// TIA Portal V20 export
VAR_GLOBAL   // PLC tag table "Unit1Em12"
   "BA060ZSIBK18.00" AT %I1068.0 : Bool;   // (HOME) WEIGHT NG CLAMP MOVER OPEN
   "BA060ZSIBK18.01" AT %I1068.1 : Bool;   // (HOME) WEIGHT NG CLAMP LEFT OPEN
   "BA060ZSIBK18.02" AT %I1068.2 : Bool;   // (HOME) WEIGHT NG CLAMP RIGHT OPEN
   "BA060ZSIBK18.03" AT %I1068.3 : Bool;   // (HOME) WEIGHT NG CLAMP Z-AXIS UP
   "BA060ZSIBK18.04" AT %I1068.4 : Bool;   // (HOME) WEIGHT NG CLAMP MOVER BACKWARD
   "BA060ZSIBK18.05" AT %I1068.5 : Bool;   // (HOME) WEIGHT NG BOX LIFT DOWN
   "BA060ZSIBK18.06" AT %I1068.6 : Bool;   // (HOME) WEIGHT NG BOX LOCK DOWN
   "BA060ZSIBK18.07" AT %I1068.7 : Bool;   // STACK NG FULL SENSOR
   "BA060ZSIBK18.08" AT %I1069.0 : Bool;   // (WORK) WEIGHT NG CLAMP MOVER CLOSE
   "BA060ZSIBK18.09" AT %I1069.1 : Bool;   // (WORK) WEIGHT NG CLAMP LEFT CLOSE
   "BA060ZSIBK18.10" AT %I1069.2 : Bool;   // (WORK) WEIGHT NG CLAMP RIGHT CLOSE
   "BA060ZSIBK18.11" AT %I1069.3 : Bool;   // (WORK) WEIGHT NG CLAMP Z-AXIS DOWN
   "BA060ZSIBK18.12" AT %I1069.4 : Bool;   // (WORK) WEIGHT NG CLAMP MOVER FORWARD
   "BA060ZSIBK18.13" AT %I1069.5 : Bool;   // (WORK) WEIGHT NG BOX LIFT UP
   "BA060ZSIBK18.14" AT %I1069.6 : Bool;   // (WORK) WEIGHT NG BOX LOCK UP
   "BA060ZSIBK18.15" AT %I1069.7 : Bool;   // SPARE
   "BA060ZSIPM10.00" AT %Q2036.0 : Bool;   // (WORK) STACK NG CLAMP MOVER CLOSE
   "BA060ZSIPM10.01" AT %Q2036.1 : Bool;   // (HOME) STACK NG CLAMP MOVER OPEN
   "BA060ZSIPM10.02" AT %Q2036.2 : Bool;   // (WORK) STACK NG CLAMP LEFT CLOSE
   "BA060ZSIPM10.03" AT %Q2036.3 : Bool;   // (HOME) STACK NG CLAMP LEFT OPEN
   "BA060ZSIPM10.04" AT %Q2036.4 : Bool;   // (WORK) STACK NG CLAMP RIGHT CLOSE
   "BA060ZSIPM10.05" AT %Q2036.5 : Bool;   // (HOME) STACK NG CLAMP RIGHT OPEN
   "BA060ZSIPM10.06" AT %Q2036.6 : Bool;   // (HOME) STACK NG CLAMP Z-AXIS UP
   "BA060ZSIPM10.07" AT %Q2036.7 : Bool;   // (WORK) STACK NG CLAMP Z-AXIS DOWN
   "BA060ZSIPM10.10" AT %Q2037.0 : Bool;   // (WORK) STACK NG CLAMP MOVER FORWARD
   "BA060ZSIPM10.11" AT %Q2037.1 : Bool;   // (HOME) STACK NG CLAMP MOVER BACKWARD
   "BA060ZSIPM10.12" AT %Q2037.2 : Bool;   // (WORK) STACK NG BOX LIFT UP
   "BA060ZSIPM10.13" AT %Q2037.3 : Bool;   // (HOME) STACK NG BOX LIFT DOWN
   "BA060ZSIPM10.14" AT %Q2037.4 : Bool;   // (WORK) STACK NG BOX LOCK UP
   "BA060ZSIPM10.15" AT %Q2037.5 : Bool;   // (HOME) STACK NG BOX LOCK DOWN
   "BA060ZSIPM10.16" AT %Q2037.6 : Bool;   // SPARE
   "BA060ZSIPM10.17" AT %Q2037.7 : Bool;   // SPARE
END_VAR
VAR_GLOBAL CONSTANT   // user constants
   U1EM12_JOB01 : DInt := 1;
   U1EM12_JOB02 : DInt := 2;
   U1EM12_JOB03 : DInt := 3;
   U1EM12_JOB04 : DInt := 4;
   U1EM12_JOB05 : DInt := 5;
   U1EM12_JOB06 : DInt := 6;
   U1EM12_JOB07 : DInt := 7;
   U1EM12_JOB08 : DInt := 8;
   U1EM12_JOB09 : DInt := 9;
   U1EM12_JOB10 : DInt := 10;
   U1EM12_JOB11 : DInt := 11;
   U1EM12_JOB12 : DInt := 12;
   U1EM12_JOB13 : DInt := 13;
   U1EM12_JOB14 : DInt := 14;
   U1EM12_JOB15 : DInt := 15;
   U1EM12_JOB16 : DInt := 16;
   U1EM12_JOB17 : DInt := 17;
   U1EM12_JOB18 : DInt := 18;
   U1EM12_JOB19 : DInt := 19;
   U1EM12_JOB20 : DInt := 20;
   U1EM12_JOB21 : DInt := 21;
   U1EM12_JOB22 : DInt := 22;
   U1EM12_JOB23 : DInt := 23;
   U1EM12_JOB24 : DInt := 24;
   U1EM12_JOB25 : DInt := 25;
   U1EM12_JOB26 : DInt := 26;
   U1EM12_JOB27 : DInt := 27;
   U1EM12_JOB28 : DInt := 28;
   U1EM12_JOB29 : DInt := 29;
   U1EM12_JOB30 : DInt := 30;
   U1EM12_JOB31 : DInt := 31;
   U1EM12_JOB32 : DInt := 32;
   U1EM12_JOB33 : DInt := 33;
   U1EM12_JOB34 : DInt := 34;
   U1EM12_JOB35 : DInt := 35;
   U1EM12_JOB36 : DInt := 36;
   U1EM12_JOB37 : DInt := 37;
   U1EM12_JOB38 : DInt := 38;
   U1EM12_JOB39 : DInt := 39;
   U1EM12_JOB40 : DInt := 40;
   U1EM12_JOB41 : DInt := 41;
   U1EM12_JOB42 : DInt := 42;
   U1EM12_JOB43 : DInt := 43;
   U1EM12_JOB44 : DInt := 44;
   U1EM12_JOB45 : DInt := 45;
   U1EM12_JOB46 : DInt := 46;
   U1EM12_JOB47 : DInt := 47;
   U1EM12_JOB48 : DInt := 48;
   U1EM12_JOB49 : DInt := 49;
   U1EM12_JOB50 : DInt := 50;
   U1EM12_JOB51 : DInt := 51;
   U1EM12_JOB52 : DInt := 52;
   U1EM12_JOB53 : DInt := 53;
   U1EM12_JOB54 : DInt := 54;
   U1EM12_JOB55 : DInt := 55;
   U1EM12_JOB56 : DInt := 56;
   U1EM12_JOB57 : DInt := 57;
   U1EM12_JOB58 : DInt := 58;
   U1EM12_JOB59 : DInt := 59;
   U1EM12_JOB60 : DInt := 60;
   U1EM12_JOB61 : DInt := 61;
   U1EM12_JOB62 : DInt := 62;
   U1EM12_JOB63 : DInt := 63;
   U1EM12_JOB64 : DInt := 64;
   U1EM12_JOB65 : DInt := 65;
   U1EM12_JOB66 : DInt := 66;
   U1EM12_JOB67 : DInt := 67;
   U1EM12_JOB68 : DInt := 68;
   U1EM12_JOB69 : DInt := 69;
   U1EM12_JOB70 : DInt := 70;
   U1EM12_JOB71 : DInt := 71;
   U1EM12_JOB72 : DInt := 72;
   U1EM12_JOB73 : DInt := 73;
   U1EM12_JOB74 : DInt := 74;
   U1EM12_JOB75 : DInt := 75;
   U1EM12_JOB76 : DInt := 76;
   U1EM12_JOB77 : DInt := 77;
   U1EM12_JOB78 : DInt := 78;
   U1EM12_JOB79 : DInt := 79;
   U1EM12_JOB80 : DInt := 80;
   U1EM12_JOB81 : DInt := 81;
   U1EM12_JOB82 : DInt := 82;
   U1EM12_JOB83 : DInt := 83;
   U1EM12_JOB84 : DInt := 84;
   U1EM12_JOB85 : DInt := 85;
   U1EM12_JOB86 : DInt := 86;
   U1EM12_JOB87 : DInt := 87;
   U1EM12_JOB88 : DInt := 88;
   U1EM12_JOB89 : DInt := 89;
   U1EM12_JOB90 : DInt := 90;
   U1EM12_JOB91 : DInt := 91;
   U1EM12_JOB92 : DInt := 92;
   U1EM12_JOB93 : DInt := 93;
   U1EM12_JOB94 : DInt := 94;
   U1EM12_JOB95 : DInt := 95;
   U1EM12_JOB96 : DInt := 96;
   U1EM12_JOB97 : DInt := 97;
   U1EM12_JOB98 : DInt := 98;
   U1EM12_JOB99 : DInt := 99;
   U1EM12_SEQUENCE01 : Int := 1;
   U1EM12_SEQUENCE02 : Int := 2;
   U1EM12_SEQUENCE03 : Int := 3;
   U1EM12_SEQUENCE04 : Int := 4;
   U1EM12_SEQUENCE05 : Int := 5;
   U1EM12_SEQUENCE06 : Int := 6;
   U1EM12_SEQUENCE07 : Int := 7;
   U1EM12_SEQUENCE08 : Int := 8;
   U1EM12_SEQUENCE09 : Int := 9;
   U1EM12_SEQUENCE10 : Int := 10;
   U1EM12_SEQUENCE11 : Int := 11;
   U1EM12_SEQUENCE12 : Int := 12;
   U1EM12_SEQUENCE13 : Int := 13;
   U1EM12_SEQUENCE14 : Int := 14;
   U1EM12_SEQUENCE15 : Int := 15;
   U1EM12_SEQUENCE16 : Int := 16;
   U1EM12_SEQUENCE17 : Int := 17;
   U1EM12_SEQUENCE18 : Int := 18;
   U1EM12_SEQUENCE19 : Int := 19;
   U1EM12_SEQUENCE20 : Int := 20;
   U1EM12_SEQUENCE21 : Int := 21;
   U1EM12_SEQUENCE22 : Int := 22;
   U1EM12_SEQUENCE23 : Int := 23;
   U1EM12_SEQUENCE24 : Int := 24;
   U1EM12_SEQUENCE25 : Int := 25;
   U1EM12_SEQUENCE26 : Int := 26;
   U1EM12_SEQUENCE27 : Int := 27;
   U1EM12_SEQUENCE28 : Int := 28;
   U1EM12_SEQUENCE29 : Int := 29;
   U1EM12_SEQUENCE30 : Int := 30;
   U1EM12_SEQUENCE31 : Int := 31;
   U1EM12_SEQUENCE32 : Int := 32;
   U1EM12_SEQUENCE33 : Int := 33;
   U1EM12_SEQUENCE34 : Int := 34;
   U1EM12_SEQUENCE35 : Int := 35;
   U1EM12_SEQUENCE36 : Int := 36;
   U1EM12_SEQUENCE37 : Int := 37;
   U1EM12_SEQUENCE38 : Int := 38;
   U1EM12_SEQUENCE39 : Int := 39;
   U1EM12_SEQUENCE40 : Int := 40;
   U1EM12_SEQUENCE41 : Int := 41;
   U1EM12_SEQUENCE42 : Int := 42;
   U1EM12_SEQUENCE43 : Int := 43;
   U1EM12_SEQUENCE44 : Int := 44;
   U1EM12_SEQUENCE45 : Int := 45;
   U1EM12_SEQUENCE46 : Int := 46;
   U1EM12_SEQUENCE47 : Int := 47;
   U1EM12_SEQUENCE48 : Int := 48;
   U1EM12_SEQUENCE49 : Int := 49;
   U1EM12_SEQUENCE50 : Int := 50;
   U1EM12_SEQUENCE51 : Int := 51;
   U1EM12_SEQUENCE52 : Int := 52;
   U1EM12_SEQUENCE53 : Int := 53;
   U1EM12_SEQUENCE54 : Int := 54;
   U1EM12_SEQUENCE55 : Int := 55;
   U1EM12_SEQUENCE56 : Int := 56;
   U1EM12_SEQUENCE57 : Int := 57;
   U1EM12_SEQUENCE58 : Int := 58;
   U1EM12_SEQUENCE59 : Int := 59;
   U1EM12_SEQUENCE60 : Int := 60;
   U1EM12_SEQUENCE61 : Int := 61;
   U1EM12_SEQUENCE62 : Int := 62;
   U1EM12_SEQUENCE63 : Int := 63;
   U1EM12_SEQUENCE64 : Int := 64;
   U1EM12_SEQUENCE65 : Int := 65;
   U1EM12_SEQUENCE66 : Int := 66;
   U1EM12_SEQUENCE67 : Int := 67;
   U1EM12_SEQUENCE68 : Int := 68;
   U1EM12_SEQUENCE69 : Int := 69;
   U1EM12_SEQUENCE70 : Int := 70;
   U1EM12_SEQUENCE71 : Int := 71;
   U1EM12_SEQUENCE72 : Int := 72;
   U1EM12_SEQUENCE73 : Int := 73;
   U1EM12_SEQUENCE74 : Int := 74;
   U1EM12_SEQUENCE75 : Int := 75;
   U1EM12_SEQUENCE76 : Int := 76;
   U1EM12_SEQUENCE77 : Int := 77;
   U1EM12_SEQUENCE78 : Int := 78;
   U1EM12_SEQUENCE79 : Int := 79;
   U1EM12_SEQUENCE80 : Int := 80;
   U1EM12_SEQUENCE81 : Int := 81;
   U1EM12_SEQUENCE82 : Int := 82;
   U1EM12_SEQUENCE83 : Int := 83;
   U1EM12_SEQUENCE84 : Int := 84;
   U1EM12_SEQUENCE85 : Int := 85;
   U1EM12_SEQUENCE86 : Int := 86;
   U1EM12_SEQUENCE87 : Int := 87;
   U1EM12_SEQUENCE88 : Int := 88;
   U1EM12_SEQUENCE89 : Int := 89;
   U1EM12_SEQUENCE90 : Int := 90;
   U1EM12_SEQUENCE91 : Int := 91;
   U1EM12_SEQUENCE92 : Int := 92;
   U1EM12_SEQUENCE93 : Int := 93;
   U1EM12_SEQUENCE94 : Int := 94;
   U1EM12_SEQUENCE95 : Int := 95;
   U1EM12_SEQUENCE96 : Int := 96;
   U1EM12_SEQUENCE97 : Int := 97;
   U1EM12_SEQUENCE98 : Int := 98;
   U1EM12_SEQUENCE99 : Int := 99;
   U1EM12_NO_OF_SEQUENCE : Int := 1;
END_VAR
